// Mitsubishi GX Developer project: Solution   PLC: FX series

PROGRAM MAIN
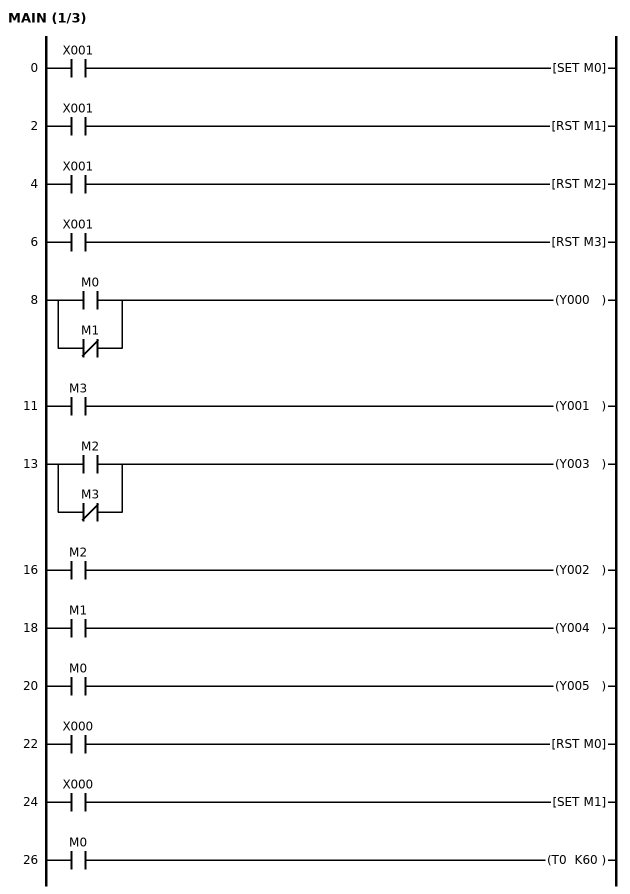
0     LD      X001
      SET     M0
2     LD      X001
      RST     M1
4     LD      X001
      RST     M2
6     LD      X001
      RST     M3
8     LD      M0
      ORI     M1
      OUT     Y000
11    LD      M3
      OUT     Y001
13    LD      M2
      ORI     M3
      OUT     Y003
16    LD      M2
      OUT     Y002
18    LD      M1
      OUT     Y004
20    LD      M0
      OUT     Y005
22    LD      X000
      RST     M0
24    LD      X000
      SET     M1
26    LD      M0
      OUT     T0 K60
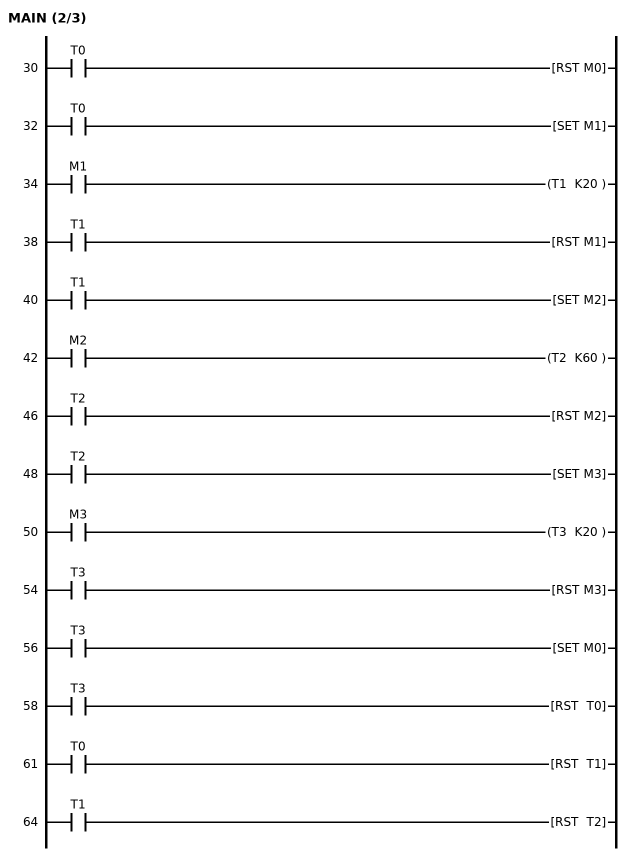
30    LD      T0
      RST     M0
32    LD      T0
      SET     M1
34    LD      M1
      OUT     T1 K20
38    LD      T1
      RST     M1
40    LD      T1
      SET     M2
42    LD      M2
      OUT     T2 K60
46    LD      T2
      RST     M2
48    LD      T2
      SET     M3
50    LD      M3
      OUT     T3 K20
54    LD      T3
      RST     M3
56    LD      T3
      SET     M0
58    LD      T3
      RST     T0
61    LD      T0
      RST     T1
64    LD      T1
      RST     T2
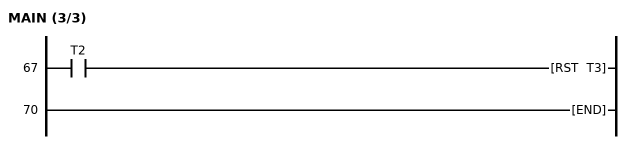
67    LD      T2
      RST     T3
70    END
END_PROGRAM
